{region '#Template'}
	{attribute 'Version' := '5.1.0.0'}
	{attribute 'Tags' := '"LCID": "1031", "Text": "Gebäudeautomation, Alarme"'}
	{attribute 'Tags' := '"LCID": "1033", "Text": "Building automation, Alarms"'}
	{attribute 'Description' := '"LCID": "1031", "Text": "Gebäude Alarme"'}
	{attribute 'Description' := '"LCID": "1033", "Text": "Building Alarms"'}
{endregion}
FUNCTION_BLOCK FB_BA_HazardDetectionAlarmSystems EXTENDS FB_BA_View
VAR_INPUT
END_VAR
VAR_OUTPUT
END_VAR
VAR_INPUT CONSTANT
	FireAlarmSystem01			: FB_BA_FireAlarmSystem;
	BurglarAlarmSystem01		: FB_BA_BurglarAlarmSystem;
END_VAR
VAR
END_VAR

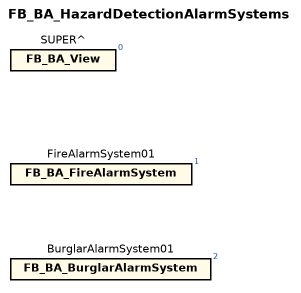
SUPER^(); // FB_BA_View
FireAlarmSystem01(); // FB_BA_FireAlarmSystem
BurglarAlarmSystem01(); // FB_BA_BurglarAlarmSystem

METHOD FB_init : BOOL
VAR_INPUT
	bInitRetains : BOOL; // if TRUE, the retain variables are initialized (warm start / cold start)
	bInCopyCode : BOOL;  // if TRUE, the instance afterwards gets moved into the copy code (online change)
END_VAR
FireAlarmSystem01.iParent			:= THIS^;	
FireAlarmSystem01.iLabel			:= LblPlt_Fire_detection_and_alarm_systems;
FireAlarmSystem01.sObjectName		:= '{Idx=61}';
FireAlarmSystem01.eDPADMode			:= E_BA_DPADMode.eInclude;

BurglarAlarmSystem01.iParent		:= THIS^;	
BurglarAlarmSystem01.iLabel			:= LblPlt_Burglar_alarm_systems;
BurglarAlarmSystem01.sObjectName	:= '{Idx=71}';
BurglarAlarmSystem01.eDPADMode		:= E_BA_DPADMode.eInclude;
END_METHOD

END_FUNCTION_BLOCK

(* stored: Version 1.1.0.1, ProductVersion 3.1.4024.12
   POU FB_BA_HazardDetectionAlarmSystems: Id {3cc02bd1-29e8-485d-8365-2550471119b9}, SpecialFunc None
   Method FB_init: Id {681ca2f1-e46a-42b1-b752-c41a2685b6c0} *)
